// TIA Portal project "Sistema Refredament" (V14)

(* hardware
DEVICE "S7-1200 station_2"  S7-1200 Station
   slot 0: "Rack_0"  S7-1200 Rack  Rack  V1.0
   slot 1: "PLC SISTEMA REFREDAMENT I VAPOR MARMITES NAU 3"  CPU 1214C DC/DC/DC  6ES7 214-1AG40-0XB0  V4.2
   slot 2: "AQ 4x14BIT_1"  6ES7 232-4HD32-0XB0  V2.0
   slot 3: "AI 8xRTD_1"  SM 1231 AI8 x RTD  6ES7 231-5PF32-0XB0  V2.0
*)

// ===== PLC "PLC SISTEMA REFREDAMENT I VAPOR MARMITES NAU 3"  CPU 1214C DC/DC/DC =====

VAR_GLOBAL   // PLC tag table "Marcas de ciclo"
   "System_Byte" AT %MB4001 : Byte;
   "FirstScan" AT %M4001.0 : Bool;
   "DiagStatusUpdate" AT %M4001.1 : Bool;
   "AlwaysTRUE" AT %M4001.2 : Bool;
   "AlwaysFALSE" AT %M4001.3 : Bool;
   "Clock_Byte" AT %MB4000 : Byte;
   "Clock_10Hz" AT %M4000.0 : Bool;
   "Clock_5Hz" AT %M4000.1 : Bool;
   "Clock_2.5Hz" AT %M4000.2 : Bool;
   "Clock_2Hz" AT %M4000.3 : Bool;
   "Clock_1.25Hz" AT %M4000.4 : Bool;
   "Clock_1Hz" AT %M4000.5 : Bool;
   "Clock_0.625Hz" AT %M4000.6 : Bool;
   "Clock_0.5Hz" AT %M4000.7 : Bool;
END_VAR

VAR_GLOBAL   // PLC tag table "PID Glicol"
   "Consigna Temperatura Glicol" AT %MW8 : Int;
   "Manual PID" AT %M16.0 : Bool;
   "Reset Error PID" AT %M16.1 : Bool;
   "Consigna PID" AT %MD18 : Real;
   "Histerisi PID" AT %MD22 : Real;
   "Ref_Obertura_Manual PID" AT %MD26 : Real;
   "Val_Obertura_% PID" AT %MW30 : Int;
END_VAR

VAR_GLOBAL   // PLC tag table "Sondes"
   "BT1 Sonda Entrada Glicol Bescanviador" AT %IW96 : Int;
   "BT2 Sonda Sortida Glicol Bescanviador" AT %IW98 : Int;
   "BT3 Sonda Entrada Aigua de Xarxa Bescanviador" AT %IW100 : Int;
   "BT4 Sonda Sortida Aigua de Xarxa Bescanviador" AT %IW102 : Int;
END_VAR

VAR_GLOBAL   // PLC tag table "Bomba Recirculació"
   "Temps Histerisi Afegir Aigua" AT %MD0 : Time;
   "Temps Fallo Caudal Bomba Recirculacio" AT %MD4 : Time;
   "Temps Fallo Nivell Agua" AT %MD10 : Time;
   "Reset Fallos" AT %M32.2 : Bool;
   "Led Termic" AT %M32.3 : Bool;
END_VAR

VAR_GLOBAL   // PLC tag table "Entrades i Sortides PLC"
   "Modul P.E" AT %I0.0 : Bool;   // Parada d'Emergencia.
   "Valvula Glicol" AT %QW128 : Int;
   "Sensor caudal Aigua Freda" AT %I1.1 : Bool;
   "Boia diposit acumulador d'aigua" AT %I1.0 : Bool;   // Circuit agua de red resfriada.
   "EV Afegir Aigua de Xarxa" AT %Q0.1 : Bool;   // Circuit agua de red resfriada.
   "Bomba Recirculacio Aigu de Xarxa" AT %Q0.0 : Bool;
   "Termic Bomba Recirculacio" AT %I1.2 : Bool;
   "Selector Habilitar Circuit" AT %I0.1 : Bool;
END_VAR

VAR_GLOBAL   // PLC tag table "Fallos"
   "Fallo Nivell Aigua" AT %M14.0 : Bool;
   "Fallo Caudal Recirculacio" AT %M14.1 : Bool;
   "Fallo Termic Bomba" AT %M14.2 : Bool;
   "Error PID" AT %M16.2 : Bool;
END_VAR

VAR_GLOBAL   // PLC tag table "Grafica Pantalla"
   "BT1 Sonda Entrada Glicol Bescanviador Grafica" AT %MW2096 : Int;
   "BT2 Sonda Sortida Glicol Bescanviador Grafica" AT %MW2098 : Int;
   "BT3 Sonda Entrada Aigua de Xarxa Bescanviador Grafica" AT %MW2100 : Int;
   "BT4 Sonda Sortida Aigua de Xarxa Bescanviador Grafica" AT %MW2102 : Int;
END_VAR

VAR_GLOBAL   // PLC tag table "Temp_Var"
   "t_histerisi" AT %MD2000 : Time;
   "t_fallo_caudal" AT %MD2004 : Time;
   "t_fallo_nivell" AT %MD2008 : Time;
END_VAR

DATA_BLOCK "Sistema Recirculacio Aigua Freda_DB"   // DB3
{ S7_Optimized_Access := 'TRUE' }
VERSION : 0.1
// stored: InstanceOfName Sistema Recirculacio Aigua Freda
"Sistema Recirculacio Aigua Freda"
BEGIN
END_DATA_BLOCK

// folder: System blocks/Program resources

DATA_BLOCK "Temps afegir aigua"   // DB2
{ S7_Optimized_Access := 'TRUE' }
AUTHOR : Simatic
FAMILY : IEC
NAME : IEC_TMR
VERSION : 1.0
// stored: InstanceOfName IEC_TIMER
"IEC_TIMER"
BEGIN
END_DATA_BLOCK

DATA_BLOCK "Timer_Fallo_Bomba_Recirculacio"   // DB4
{ S7_Optimized_Access := 'TRUE' }
AUTHOR : Simatic
FAMILY : IEC
NAME : IEC_TMR
VERSION : 1.0
// stored: InstanceOfName IEC_TIMER
"IEC_TIMER"
BEGIN
END_DATA_BLOCK

DATA_BLOCK "Timer Fallo Nivell Agua"   // DB5
{ S7_Optimized_Access := 'TRUE' }
AUTHOR : Simatic
FAMILY : IEC
NAME : IEC_TMR
VERSION : 1.0
// stored: InstanceOfName IEC_TIMER
"IEC_TIMER"
BEGIN
END_DATA_BLOCK

// folder: (top level)

FUNCTION_BLOCK "Sistema Recirculacio Aigua Freda"   // FB1, LAD
{ S7_Optimized_Access := 'TRUE' }
VERSION : 0.1
   VAR_INPUT
      "Marxa/Paro" : Bool;
      Seguretat : Bool;
      "Reset Fallos" : Bool;
      Termic : Bool;
      Nivell : Bool;
      "BF1 Sensor caudal Aigua Freda" : Bool;
      "Temps Histerisi Afegir Aigua" : Time := T#15s;
      "Timer Fallo Caudal Bomba Recirculacio" : Time := T#30s;
      "Timer Fallo Nivell Agua" : Time := T#10m;
   END_VAR
   VAR_OUTPUT
      Bomba : Bool;
      "EV5 Afegir Aigua de Xarxa" : Bool;
      "Fallo Termic" : Bool;
      "Fallo Caudal Recirculacio" : Bool;
      "Fallo Nivell Aigua" : Bool;
   END_VAR
   VAR
      M_Afegir_Aigua : Bool;
      "Parada per Error" : Bool;
      Flank_1 : Bool;
      Flank_2 : Bool;
      Flank_3 : Bool;
      My_INT : Int;
   END_VAR
   VAR_TEMP
      Temp_TIME : Time;
   END_VAR
   VAR_TEMP   // added for the SCL form of the ladder/FBD networks
      _w1 : Bool;
   END_VAR
BEGIN

REGION Network 1: Marxa Bomba
   // Retard de arranc de la bomba son 10s
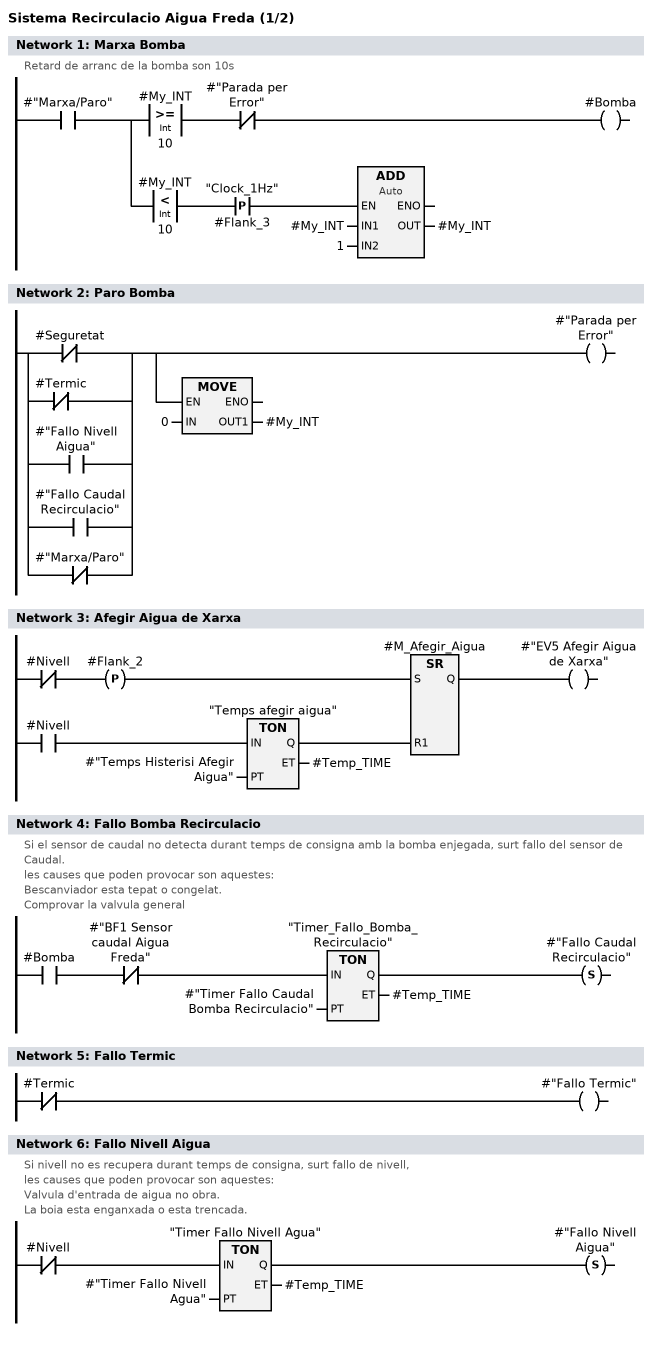
   RUNG wire#powerrail
      Contact( #"Marxa/Paro" )
      wire#w1
      { S7_Templates := "SrcType := Int" } GE_Contact(in1 := #My_INT, in2 := 10)
      I_Contact( #"Parada per Error" )
      Coil( #Bomba )
   END_RUNG
   RUNG wire#w1
      { S7_Templates := "SrcType := Int" } LT_Contact(in1 := #My_INT, in2 := 10)
      P_Contact(operand := "Clock_1Hz", bit := #Flank_3)
      Add(in1 := #My_INT, in2 := 1, out => #My_INT)
   END_RUNG
   // the same network as SCL:
   #Bomba := #"Marxa/Paro" AND (#My_INT >= 10) AND NOT #"Parada per Error";
   #_w1 := #"Marxa/Paro" AND (#My_INT < 10) AND "Clock_1Hz" AND NOT #Flank_3;   // rising edge of "Clock_1Hz"
   #Flank_3 := "Clock_1Hz";
   IF #_w1 THEN #My_INT := #My_INT + 1; END_IF;
END_REGION

REGION Network 2: Paro Bomba
   RUNG wire#powerrail
      I_Contact( #Seguretat )
      wire#w1
      Coil( #"Parada per Error" )
   END_RUNG
   RUNG wire#powerrail
      I_Contact( #Termic )
   END_RUNG wire#w1
   RUNG wire#powerrail
      Contact( #"Fallo Nivell Aigua" )
   END_RUNG wire#w1
   RUNG wire#powerrail
      Contact( #"Fallo Caudal Recirculacio" )
   END_RUNG wire#w1
   RUNG wire#powerrail
      I_Contact( #"Marxa/Paro" )
   END_RUNG wire#w1
   RUNG wire#w1
      Move(in := 0, out1 => #My_INT)
   END_RUNG
   // the same network as SCL:
   #"Parada per Error" := NOT #Seguretat OR NOT #Termic OR #"Fallo Nivell Aigua" OR #"Fallo Caudal Recirculacio" OR NOT #"Marxa/Paro";
   IF #"Parada per Error" THEN #My_INT := 0; END_IF;
END_REGION

REGION Network 3: Afegir Aigua de Xarxa
   #_w1 := NOT #Nivell AND NOT #Flank_2;   // rising edge
   #Flank_2 := NOT #Nivell;
   "Temps afegir aigua".TON(IN := #Nivell, PT := #"Temps Histerisi Afegir Aigua", ET => #Temp_TIME);
   IF #_w1 THEN
       #M_Afegir_Aigua := TRUE;   // SR flip-flop
   END_IF;
   IF "Temps afegir aigua".Q THEN #M_Afegir_Aigua := FALSE; END_IF;
   #"EV5 Afegir Aigua de Xarxa" := #M_Afegir_Aigua;
END_REGION

REGION Network 4: Fallo Bomba Recirculacio
   // Si el sensor de caudal no detecta durant temps de consigna amb la bomba enjegada, surt fallo del sensor de Caudal. 
   // 
   // les causes que poden provocar son aquestes:
   // 
   // Bescanviador esta tepat o congelat.
   // Comprovar la valvula general
   "Timer_Fallo_Bomba_Recirculacio".TON(IN := #Bomba AND NOT #"BF1 Sensor caudal Aigua Freda",
                           PT := #"Timer Fallo Caudal Bomba Recirculacio",
                           ET => #Temp_TIME);
   IF "Timer_Fallo_Bomba_Recirculacio".Q THEN #"Fallo Caudal Recirculacio" := TRUE; END_IF;
END_REGION

REGION Network 5: Fallo Termic
   RUNG wire#powerrail
      I_Contact( #Termic )
      Coil( #"Fallo Termic" )
   END_RUNG
   // the same network as SCL:
   #"Fallo Termic" := NOT #Termic;
END_REGION

REGION Network 6: Fallo Nivell Aigua
   // Si nivell no es recupera durant temps de consigna, surt fallo de nivell, 
   // 
   // les causes que poden provocar son aquestes:
   // 
   // Valvula d'entrada de aigua no obra.
   // La boia esta enganxada o esta trencada.
   "Timer Fallo Nivell Agua".TON(IN := NOT #Nivell, PT := #"Timer Fallo Nivell Agua", ET => #Temp_TIME);
   IF "Timer Fallo Nivell Agua".Q THEN #"Fallo Nivell Aigua" := TRUE; END_IF;
END_REGION

REGION Network 7: Reset Fallos
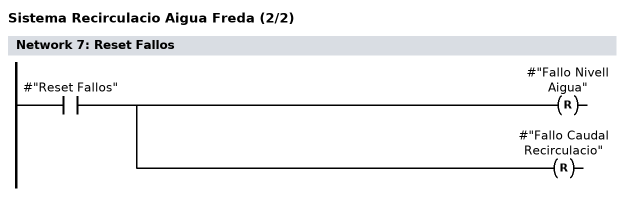
   RUNG wire#powerrail
      Contact( #"Reset Fallos" )
      wire#w1
      R_Coil( #"Fallo Nivell Aigua" )
   END_RUNG
   RUNG wire#w1
      R_Coil( #"Fallo Caudal Recirculacio" )
   END_RUNG
   // the same network as SCL:
   IF #"Reset Fallos" THEN
       #"Fallo Nivell Aigua" := FALSE;
       #"Fallo Caudal Recirculacio" := FALSE;
   END_IF;
END_REGION
END_FUNCTION_BLOCK

FUNCTION_BLOCK "Control Valvules Bascanviador"   // FB2, LAD
{ S7_Optimized_Access := 'TRUE' }
VERSION : 0.1
   VAR_INPUT
      "Clock 1 Hz" : Bool;
      "AUTO/MAN" : Bool;
      "Consigna Aigua Refredament" : Int;
      Histerisi : Int := 0;
      "Valor Manual Obertura EV1" : SInt;
      "Valor Manual Obertura EV2" : SInt;
      "Valor Manual Obertura EV3" : SInt;
      "Valor Manual Obertura EV4" : SInt;
      "Tº BT1 Sonda Entrada Glicol Bescanviador" : Int;   // -50ºC/50ºC
      "Tº BT2 Sonda Sortida Glicol Bescanviador" : Int;   // -50ºC/50ºC
      "Tº BT3 Sonda Entrada Aigua de Xarxa Bescanviador" : Int;   // -50ºC/50ºC
      "Tº BT4 Sonda Sortida Aigua de Xarxa Bescanviador" : Int;   // -50ºC/50ºC
      "Feedback EV1 Entrada Bescanviador Glicol_1" : Int;   // 4..20mA
      "Feedback EV2 Sortida Bescanviador Glicol_1" : Int;   // 4..20mA
      "Feedback EV3 Entrada Bescanviador Aigua de Xarxa_1" : Int;   // 4..20mA
      "Feedback EV4 Sortida Bescanviador Aigua de Xarxa_1" : Int;   // 4..20mA
   END_VAR
   VAR_OUTPUT
      "EV1 Entrada Bescanviador Glicol" : Int;   // 4..20mA
      "EV2 Sortida Bescanviador Glicol" : Int;   // 4..20mA
      "EV3 Entrada Bescanviador Aigua de Xarxa" : Int;   // 4..20mA
      "EV4 Sortida Bescanviador Aigua de Xarxa" : Int;   // 4..20mA
   END_VAR
   VAR
      "Impuls 1s" : Bool;
      Flank_Impuls : Bool;
      Temp_Low_Limit : Int;
      Temp_High_Limit : Int;
      Histerisis_Limited : Int;
      "Consigna Limit MIN" : Int;
      "Consigna Limit MAX" : Int;
   END_VAR
   VAR_TEMP
      "Temp BOOL" : Bool;
      "Temp INT" : Int;
      "Temp REAL" : Real;
   END_VAR
   VAR_TEMP   // added for the SCL form of the ladder/FBD networks
      _w1 : Bool;
   END_VAR
BEGIN

REGION Network 1: Impuls cada segon
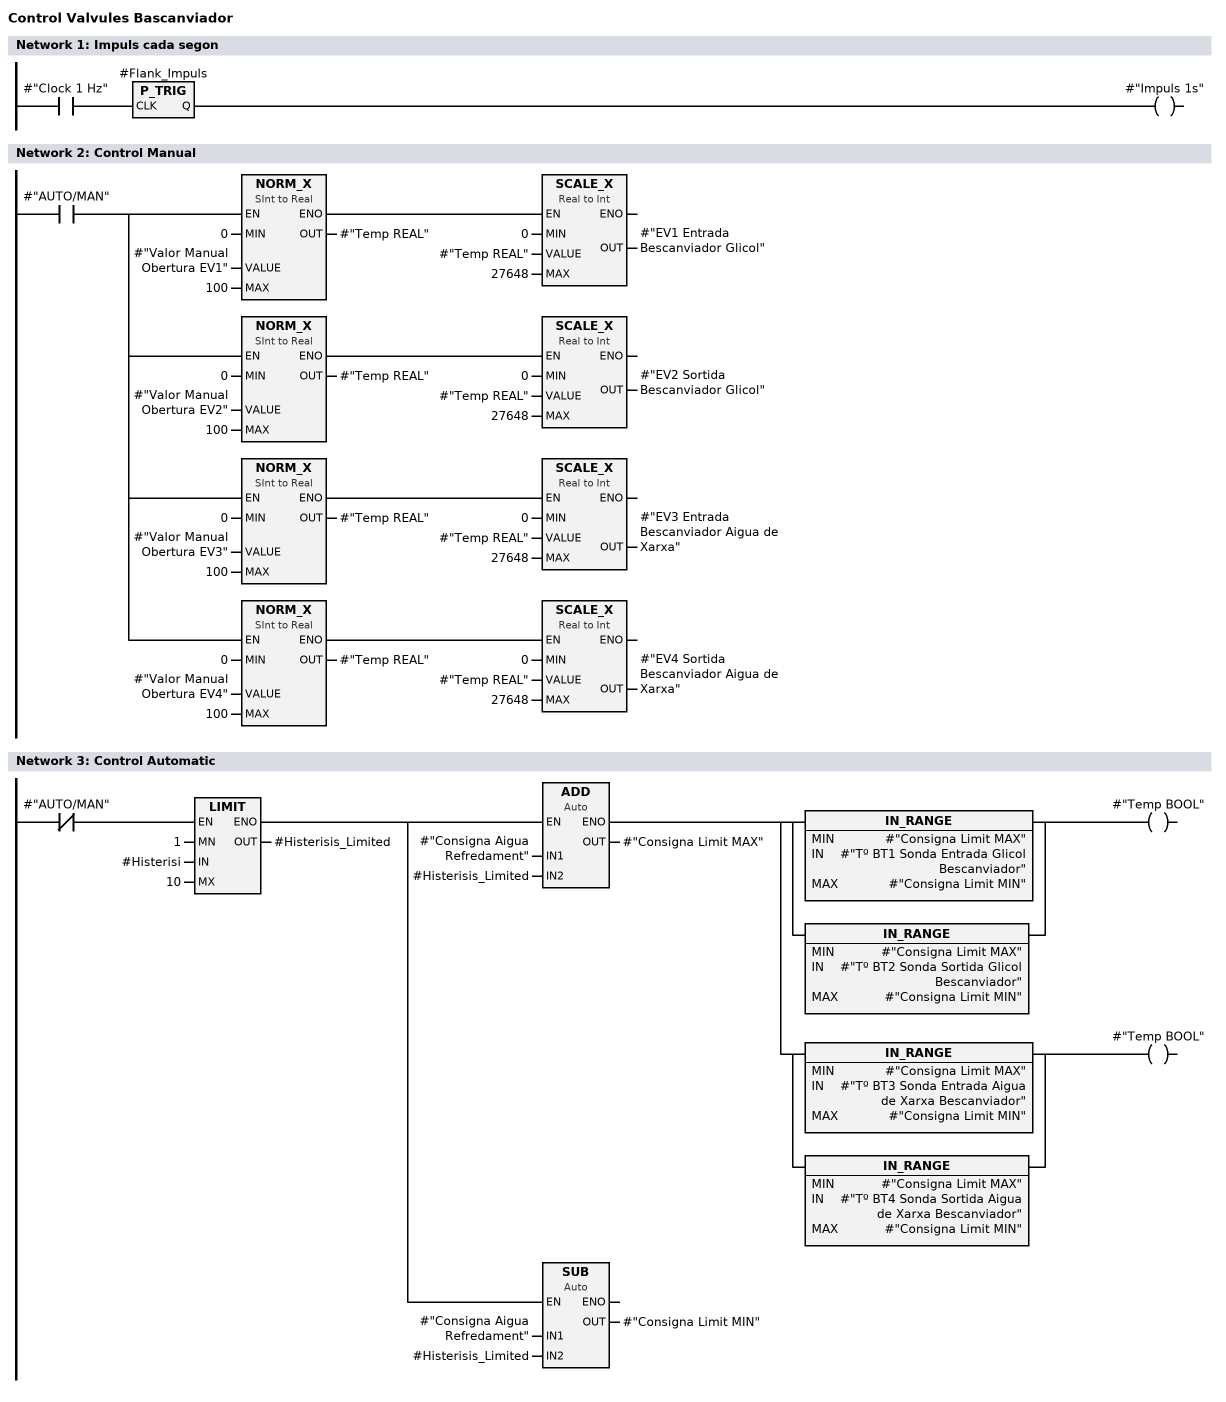
   RUNG wire#powerrail
      Contact( #"Clock 1 Hz" )
      P_Trig( #Flank_Impuls )
      Coil( #"Impuls 1s" )
   END_RUNG
   // the same network as SCL:
   #_w1 := #"Clock 1 Hz" AND NOT #Flank_Impuls;   // rising edge
   #Flank_Impuls := #"Clock 1 Hz";
   #"Impuls 1s" := #_w1;
END_REGION

REGION Network 2: Control Manual
   RUNG wire#powerrail
      Contact( #"AUTO/MAN" )
      wire#w1
      { S7_Templates := "[SrcType := SInt, DestType := Real]" } Normalize(min := 0, value := #"Valor Manual Obertura EV1", max := 100, out => #"Temp REAL")
      { S7_Templates := "[SrcType := Real, DestType := Int]" } Scale(min := 0, value := #"Temp REAL", max := 27648, out => #"EV1 Entrada Bescanviador Glicol")
   END_RUNG
   RUNG wire#w1
      { S7_Templates := "[SrcType := SInt, DestType := Real]" } Normalize(min := 0, value := #"Valor Manual Obertura EV2", max := 100, out => #"Temp REAL")
      { S7_Templates := "[SrcType := Real, DestType := Int]" } Scale(min := 0, value := #"Temp REAL", max := 27648, out => #"EV2 Sortida Bescanviador Glicol")
   END_RUNG
   RUNG wire#w1
      { S7_Templates := "[SrcType := SInt, DestType := Real]" } Normalize(min := 0, value := #"Valor Manual Obertura EV3", max := 100, out => #"Temp REAL")
      { S7_Templates := "[SrcType := Real, DestType := Int]" } Scale(min := 0, value := #"Temp REAL", max := 27648, out => #"EV3 Entrada Bescanviador Aigua de Xarxa")
   END_RUNG
   RUNG wire#w1
      { S7_Templates := "[SrcType := SInt, DestType := Real]" } Normalize(min := 0, value := #"Valor Manual Obertura EV4", max := 100, out => #"Temp REAL")
      { S7_Templates := "[SrcType := Real, DestType := Int]" } Scale(min := 0, value := #"Temp REAL", max := 27648, out => #"EV4 Sortida Bescanviador Aigua de Xarxa")
   END_RUNG
   // the same network as SCL:
   IF #"AUTO/MAN" THEN
       #"Temp REAL" := NORM_X(MIN := 0, VALUE := #"Valor Manual Obertura EV1", MAX := 100);
       #"EV1 Entrada Bescanviador Glicol" := SCALE_X(MIN := 0, VALUE := #"Temp REAL", MAX := 27648);
       #"Temp REAL" := NORM_X(MIN := 0, VALUE := #"Valor Manual Obertura EV2", MAX := 100);
       #"EV2 Sortida Bescanviador Glicol" := SCALE_X(MIN := 0, VALUE := #"Temp REAL", MAX := 27648);
       #"Temp REAL" := NORM_X(MIN := 0, VALUE := #"Valor Manual Obertura EV3", MAX := 100);
       #"EV3 Entrada Bescanviador Aigua de Xarxa" := SCALE_X(MIN := 0, VALUE := #"Temp REAL", MAX := 27648);
       #"Temp REAL" := NORM_X(MIN := 0, VALUE := #"Valor Manual Obertura EV4", MAX := 100);
       #"EV4 Sortida Bescanviador Aigua de Xarxa" := SCALE_X(MIN := 0, VALUE := #"Temp REAL", MAX := 27648);
   END_IF;
END_REGION

REGION Network 3: Control Automatic
   IF NOT #"AUTO/MAN" THEN
       #Histerisis_Limited := LIMIT(MN := 1, IN := #Histerisi, MX := 10);
       #"Consigna Limit MAX" := #"Consigna Aigua Refredament" + #Histerisis_Limited;
   END_IF;
   #"Temp BOOL" := NOT #"AUTO/MAN" AND (((#"Consigna Limit MAX" <= #"Tº BT1 Sonda Entrada Glicol Bescanviador") AND (#"Tº BT1 Sonda Entrada Glicol Bescanviador" <= #"Consigna Limit MIN")) OR ((#"Consigna Limit MAX" <= #"Tº BT2 Sonda Sortida Glicol Bescanviador") AND (#"Tº BT2 Sonda Sortida Glicol Bescanviador" <= #"Consigna Limit MIN")));
   #"Temp BOOL" := NOT #"AUTO/MAN" AND (((#"Consigna Limit MAX" <= #"Tº BT3 Sonda Entrada Aigua de Xarxa Bescanviador") AND (#"Tº BT3 Sonda Entrada Aigua de Xarxa Bescanviador" <= #"Consigna Limit MIN")) OR ((#"Consigna Limit MAX" <= #"Tº BT4 Sonda Sortida Aigua de Xarxa Bescanviador") AND (#"Tº BT4 Sonda Sortida Aigua de Xarxa Bescanviador" <= #"Consigna Limit MIN")));
   IF NOT #"AUTO/MAN" THEN
       #"Consigna Limit MIN" := #"Consigna Aigua Refredament" - #Histerisis_Limited;
   END_IF;
END_REGION
END_FUNCTION_BLOCK

FUNCTION "Obertura de valvules amb percentatge" : Void   // FC1, LAD
{ S7_Optimized_Access := 'TRUE' }
VERSION : 0.1
   VAR_INPUT
      IN : Int;
   END_VAR
   VAR_OUTPUT
      OUT : Int;
   END_VAR
   VAR_TEMP
      Temp_REAL : Real;
   END_VAR
BEGIN

REGION Network 1
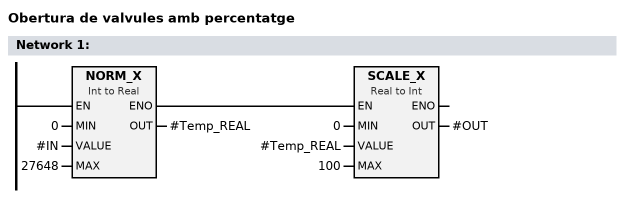
   RUNG wire#powerrail
      { S7_Templates := "[SrcType := Int, DestType := Real]" } Normalize(min := 0, value := #IN, max := 27648, out => #Temp_REAL)
      { S7_Templates := "[SrcType := Real, DestType := Int]" } Scale(min := 0, value := #Temp_REAL, max := 100, out => #OUT)
   END_RUNG
   // the same network as SCL:
   #Temp_REAL := NORM_X(MIN := 0, VALUE := #IN, MAX := 27648);
   #OUT := SCALE_X(MIN := 0, VALUE := #Temp_REAL, MAX := 100);
END_REGION
END_FUNCTION

ORGANIZATION_BLOCK "Main"   // OB1, LAD, ProgramCycle
TITLE = "Main Program Sweep (Cycle)"
{ S7_Optimized_Access := 'TRUE' }
VERSION : 0.1
   VAR_INPUT
      Initial_Call : Bool;   // Initial call of this OB
      Remanence : Bool;   // =True, if remanent data are available
   END_VAR
   VAR_TEMP
      Temp_REAL : Real;
      "% Obertura" : SInt;
   END_VAR
BEGIN

REGION Network 1: Bomba Recirculacio
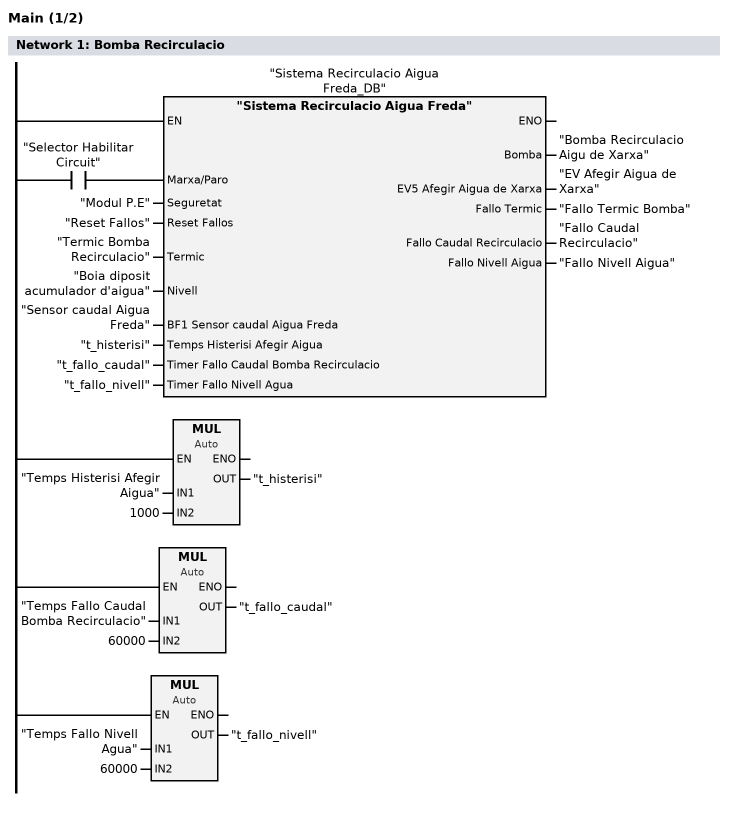
   RUNG wire#powerrail
      "Sistema Recirculacio Aigua Freda_DB"("Marxa/Paro" := wire#w1, Seguretat := "Modul P.E", "Reset Fallos" := "Reset Fallos", Termic := "Termic Bomba Recirculacio", Nivell := "Boia diposit acumulador d'aigua", "BF1 Sensor caudal Aigua Freda" := "Sensor caudal Aigua Freda", "Temps Histerisi Afegir Aigua" := "t_histerisi", "Timer Fallo Caudal Bomba Recirculacio" := "t_fallo_caudal", "Timer Fallo Nivell Agua" := "t_fallo_nivell", Bomba => "Bomba Recirculacio Aigu de Xarxa", "EV5 Afegir Aigua de Xarxa" => "EV Afegir Aigua de Xarxa", "Fallo Termic" => "Fallo Termic Bomba", "Fallo Caudal Recirculacio" => "Fallo Caudal Recirculacio", "Fallo Nivell Aigua" => "Fallo Nivell Aigua")
   END_RUNG
   RUNG wire#powerrail
      Contact( "Selector Habilitar Circuit" )
   END_RUNG wire#w1
   RUNG wire#powerrail
      Mul(in1 := "Temps Histerisi Afegir Aigua", in2 := 1000, out => "t_histerisi")
   END_RUNG
   RUNG wire#powerrail
      Mul(in1 := "Temps Fallo Caudal Bomba Recirculacio", in2 := 60000, out => "t_fallo_caudal")
   END_RUNG
   RUNG wire#powerrail
      Mul(in1 := "Temps Fallo Nivell Agua", in2 := 60000, out => "t_fallo_nivell")
   END_RUNG
   // the same network as SCL:
   "Sistema Recirculacio Aigua Freda_DB"("Marxa/Paro" := "Selector Habilitar Circuit",   // "Sistema Recirculacio Aigua Freda"
                           Seguretat := "Modul P.E",
                           "Reset Fallos" := "Reset Fallos",
                           Termic := "Termic Bomba Recirculacio",
                           Nivell := "Boia diposit acumulador d'aigua",
                           "BF1 Sensor caudal Aigua Freda" := "Sensor caudal Aigua Freda",
                           "Temps Histerisi Afegir Aigua" := "t_histerisi",
                           "Timer Fallo Caudal Bomba Recirculacio" := "t_fallo_caudal",
                           "Timer Fallo Nivell Agua" := "t_fallo_nivell",
                           Bomba => "Bomba Recirculacio Aigu de Xarxa",
                           "EV5 Afegir Aigua de Xarxa" => "EV Afegir Aigua de Xarxa",
                           "Fallo Termic" => "Fallo Termic Bomba",
                           "Fallo Caudal Recirculacio" => "Fallo Caudal Recirculacio",
                           "Fallo Nivell Aigua" => "Fallo Nivell Aigua");
   "t_histerisi" := "Temps Histerisi Afegir Aigua" * 1000;
   "t_fallo_caudal" := "Temps Fallo Caudal Bomba Recirculacio" * 60000;
   "t_fallo_nivell" := "Temps Fallo Nivell Agua" * 60000;
END_REGION

REGION Network 2: Grafica Pantalla
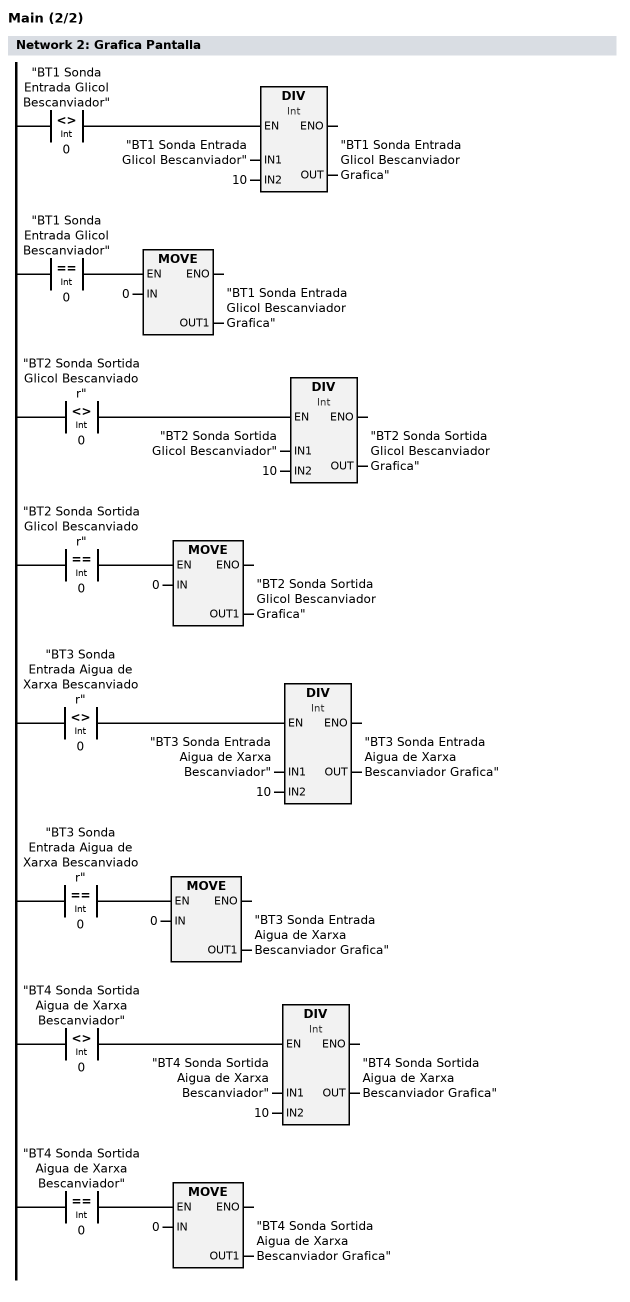
   RUNG wire#powerrail
      { S7_Templates := "SrcType := Int" } NE_Contact(in1 := "BT1 Sonda Entrada Glicol Bescanviador", in2 := 0)
      { S7_Templates := "SrcType := Int" } Div(in1 := "BT1 Sonda Entrada Glicol Bescanviador", in2 := 10, out => "BT1 Sonda Entrada Glicol Bescanviador Grafica")
   END_RUNG
   RUNG wire#powerrail
      { S7_Templates := "SrcType := Int" } EQ_Contact(in1 := "BT1 Sonda Entrada Glicol Bescanviador", in2 := 0)
      Move(in := 0, out1 => "BT1 Sonda Entrada Glicol Bescanviador Grafica")
   END_RUNG
   RUNG wire#powerrail
      { S7_Templates := "SrcType := Int" } NE_Contact(in1 := "BT2 Sonda Sortida Glicol Bescanviador", in2 := 0)
      { S7_Templates := "SrcType := Int" } Div(in1 := "BT2 Sonda Sortida Glicol Bescanviador", in2 := 10, out => "BT2 Sonda Sortida Glicol Bescanviador Grafica")
   END_RUNG
   RUNG wire#powerrail
      { S7_Templates := "SrcType := Int" } EQ_Contact(in1 := "BT2 Sonda Sortida Glicol Bescanviador", in2 := 0)
      Move(in := 0, out1 => "BT2 Sonda Sortida Glicol Bescanviador Grafica")
   END_RUNG
   RUNG wire#powerrail
      { S7_Templates := "SrcType := Int" } NE_Contact(in1 := "BT3 Sonda Entrada Aigua de Xarxa Bescanviador", in2 := 0)
      { S7_Templates := "SrcType := Int" } Div(in1 := "BT3 Sonda Entrada Aigua de Xarxa Bescanviador", in2 := 10, out => "BT3 Sonda Entrada Aigua de Xarxa Bescanviador Grafica")
   END_RUNG
   RUNG wire#powerrail
      { S7_Templates := "SrcType := Int" } EQ_Contact(in1 := "BT3 Sonda Entrada Aigua de Xarxa Bescanviador", in2 := 0)
      Move(in := 0, out1 => "BT3 Sonda Entrada Aigua de Xarxa Bescanviador Grafica")
   END_RUNG
   RUNG wire#powerrail
      { S7_Templates := "SrcType := Int" } NE_Contact(in1 := "BT4 Sonda Sortida Aigua de Xarxa Bescanviador", in2 := 0)
      { S7_Templates := "SrcType := Int" } Div(in1 := "BT4 Sonda Sortida Aigua de Xarxa Bescanviador", in2 := 10, out => "BT4 Sonda Sortida Aigua de Xarxa Bescanviador Grafica")
   END_RUNG
   RUNG wire#powerrail
      { S7_Templates := "SrcType := Int" } EQ_Contact(in1 := "BT4 Sonda Sortida Aigua de Xarxa Bescanviador", in2 := 0)
      Move(in := 0, out1 => "BT4 Sonda Sortida Aigua de Xarxa Bescanviador Grafica")
   END_RUNG
   // the same network as SCL:
   IF "BT1 Sonda Entrada Glicol Bescanviador" <> 0 THEN
       "BT1 Sonda Entrada Glicol Bescanviador Grafica" := "BT1 Sonda Entrada Glicol Bescanviador" / 10;
   END_IF;
   IF "BT1 Sonda Entrada Glicol Bescanviador" = 0 THEN
       "BT1 Sonda Entrada Glicol Bescanviador Grafica" := 0;
   END_IF;
   IF "BT2 Sonda Sortida Glicol Bescanviador" <> 0 THEN
       "BT2 Sonda Sortida Glicol Bescanviador Grafica" := "BT2 Sonda Sortida Glicol Bescanviador" / 10;
   END_IF;
   IF "BT2 Sonda Sortida Glicol Bescanviador" = 0 THEN
       "BT2 Sonda Sortida Glicol Bescanviador Grafica" := 0;
   END_IF;
   IF "BT3 Sonda Entrada Aigua de Xarxa Bescanviador" <> 0 THEN
       "BT3 Sonda Entrada Aigua de Xarxa Bescanviador Grafica" := "BT3 Sonda Entrada Aigua de Xarxa Bescanviador" / 10;
   END_IF;
   IF "BT3 Sonda Entrada Aigua de Xarxa Bescanviador" = 0 THEN
       "BT3 Sonda Entrada Aigua de Xarxa Bescanviador Grafica" := 0;
   END_IF;
   IF "BT4 Sonda Sortida Aigua de Xarxa Bescanviador" <> 0 THEN
       "BT4 Sonda Sortida Aigua de Xarxa Bescanviador Grafica" := "BT4 Sonda Sortida Aigua de Xarxa Bescanviador" / 10;
   END_IF;
   IF "BT4 Sonda Sortida Aigua de Xarxa Bescanviador" = 0 THEN
       "BT4 Sonda Sortida Aigua de Xarxa Bescanviador Grafica" := 0;
   END_IF;
END_REGION
END_ORGANIZATION_BLOCK

ORGANIZATION_BLOCK "Cyclic interrupt"   // OB30, LAD, CyclicInterrupt
{ S7_Optimized_Access := 'TRUE' }
VERSION : 0.1
   VAR_INPUT
      Initial_Call : Bool;   // Initial call of this OB
      Event_Count : Int;   // Events discarded
   END_VAR
   VAR_TEMP
      Output : Real;
      State : Int;
      Error : Bool;
      ErrorBits : DWord;
      ScaledInput : Real;
      Output_PER : Int;
      Temp_REAL : Real;
   END_VAR
BEGIN

REGION Network 1: Control Glicol
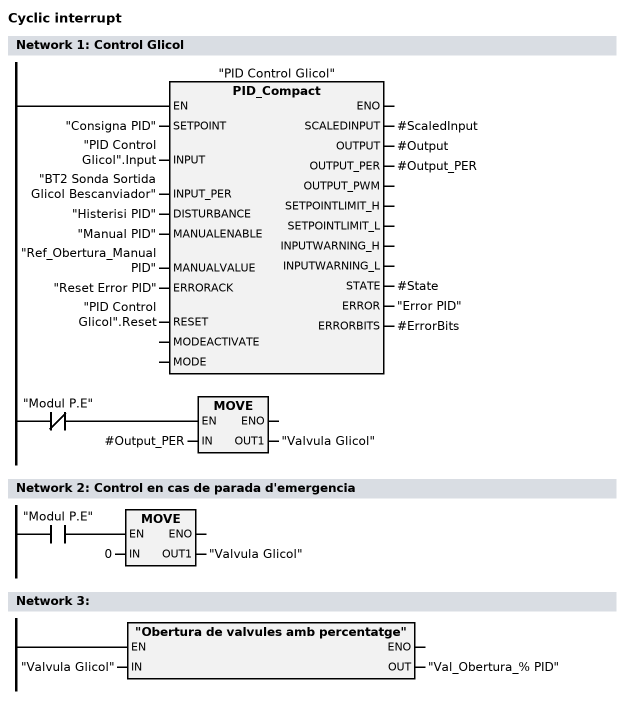
   "PID Control Glicol"(Setpoint := "Consigna PID",   // PID_Compact
                        Input := "PID Control Glicol".Input,
                        Input_PER := "BT2 Sonda Sortida Glicol Bescanviador",
                        Disturbance := "Histerisi PID",
                        ManualEnable := "Manual PID",
                        ManualValue := "Ref_Obertura_Manual PID",
                        ErrorAck := "Reset Error PID",
                        Reset := "PID Control Glicol".Reset,
                        ScaledInput => #ScaledInput,
                        Output => #Output,
                        Output_PER => #Output_PER,
                        State => #State,
                        Error => "Error PID",
                        ErrorBits => #ErrorBits);
   IF NOT "Modul P.E" THEN "Valvula Glicol" := #Output_PER; END_IF;
END_REGION

REGION Network 2: Control en cas de parada d'emergencia
   RUNG wire#powerrail
      Contact( "Modul P.E" )
      Move(in := 0, out1 => "Valvula Glicol")
   END_RUNG
   // the same network as SCL:
   IF "Modul P.E" THEN "Valvula Glicol" := 0; END_IF;
END_REGION

REGION Network 3
   RUNG wire#powerrail
      "Obertura de valvules amb percentatge"(IN := "Valvula Glicol", OUT => "Val_Obertura_% PID")
   END_RUNG
   // the same network as SCL:
   "Obertura de valvules amb percentatge"(IN := "Valvula Glicol", OUT => "Val_Obertura_% PID");
END_REGION
END_ORGANIZATION_BLOCK